// TIA Portal V18 export
TYPE "LGasp_typeRigheEliminate"
// stored: IsFailsafeCompliant false
   STRUCT
      ID : DInt;
      pzfatti : DInt;
   END_STRUCT;
END_TYPE
